// TIA Portal V18 export
FUNCTION_BLOCK "axis_FBD"   // FB53, FBD
{ S7_Optimized_Access := 'TRUE' }
VERSION : 0.1
// stored: AutoNumber true, IsIECCheckEnabled false, IsRetainMemResEnabled false, MemoryReserve 100, SetENOAutomatically false, UDAEnableTagReadback false
   VAR_INPUT
      "mm_per_ reductur outputshaft_rev (AskURmechEngineer)" : Real := 10.0;
      "reduction_ rotation (AskURmechEngineer)" : Real := 1.0;
      "ABincrements_per_ encoder_rev (CheckEnc Label and HSC hardware settings dont forget input filtration)" : Real := 4096.0;
      "max_revs_ at_10V (CheckMotorLabel)" : Real := 1360.0;
      "enc_placed_ on_motor not reductor output shaft(visually inspect)" : Bool;
      "isMultiturn (visually inspect)" : Bool;
      MultiTurnGoesFwdOnly : Bool;
      soft_speed_change_req : Bool;
      ENC_REVERSED_DIR : Bool;
      ENCODER_DINT : DInt;
      TargetUnison : Real;
      TargetHome : Real;
      Desk_bHome : Bool;
      Desk_bFwd : Bool;
      Desk_bRev : Bool;
      s_fwd_mechOK : Bool;
      s_rev_mecOK : Bool;
      s_fwd_ind : Bool;
      s_rev_ind : Bool;
      xPredifCal : Bool;
      ALIEN_MODE_EN : Bool;
      ALIEN_FWD : Bool;
      ALIEN_REV : Bool;
      ALIEN_SPDABS : Real;
      ExecUni : Bool;
      TheseAreDoors : Bool;
      xOverrideLocal : Bool;
      hbStepPlus : Bool;
      hbStepMinus : Bool;
      TargetStep : Real;
      динамические_границы_используются : Bool;
      динамическая_граница_fwd : Real;
      динамическая_граница_rev : Real;
   END_VAR
   VAR_OUTPUT
      max_speed_10V_p_mm : Real;
      speed_V : Real;
      speed : Real;
      yaINTSPEED : Int;
      yFWD : Bool;
      yREV : Bool;
      yFwd_STOP : Bool;
      yRev_STOP : Bool;
      yIN_POS : Bool;
      ER : Bool;
      WN : Bool;
      ALLOWED : Bool;
      "dist_stop(check t_acc)" : Real;
      MovingHomeWhileFree : Bool;
      ERWSTRING : WString;
   END_VAR
   VAR_IN_OUT
      aut_target : Real;
      para : "typeMotPara";
      POS : Real;
      calibrated : Bool;
      ENC_RET : "typePOSMEMcalib";
   END_VAR
   VAR
      para_ArtLimits { ExternalAccessible := 'False'; ExternalVisible := 'False'; ExternalWritable := 'False'} : "typeMotPara";
      v_absMax : Real;
      au_execute : Bool;
      AMANGRDB { S7_SetPoint := 'True'} : "axis_manager";
      MOTDB { S7_SetPoint := 'True'} : "__mot_universal_";
      WNDB { S7_SetPoint := 'True'} : "ER_WORD";
      ERDB { S7_SetPoint := 'True'} : "ER_WORD";
      erw_calcspd : WString;
      hmiResetCalib : Bool;
      IEC_Timer_0_Instance { S7_SetPoint := 'True'} : TON_TIME;
      artLimiter_Instance { S7_SetPoint := 'True'} : "artLimiter";
   END_VAR
   VAR_TEMP
      counts_per_mm : Real;
      er_params_mech : Bool;
      ENC : DInt;
      selected_man_speed : Real;
      AUTO : Bool;
      MAN : Bool;
      OVERRIDE : Bool;
      counts_real : Real;
      Enc_real_mm : Real;
      er_follow : Bool;
      er_set : Bool;
      er_fwd : Bool;
      er_rev : Bool;
      partners_calibrated : Bool;
      Selected_speed_auto : Real;
      ошибка_динамических_границ : Bool;
   END_VAR
BEGIN

REGION Network 1
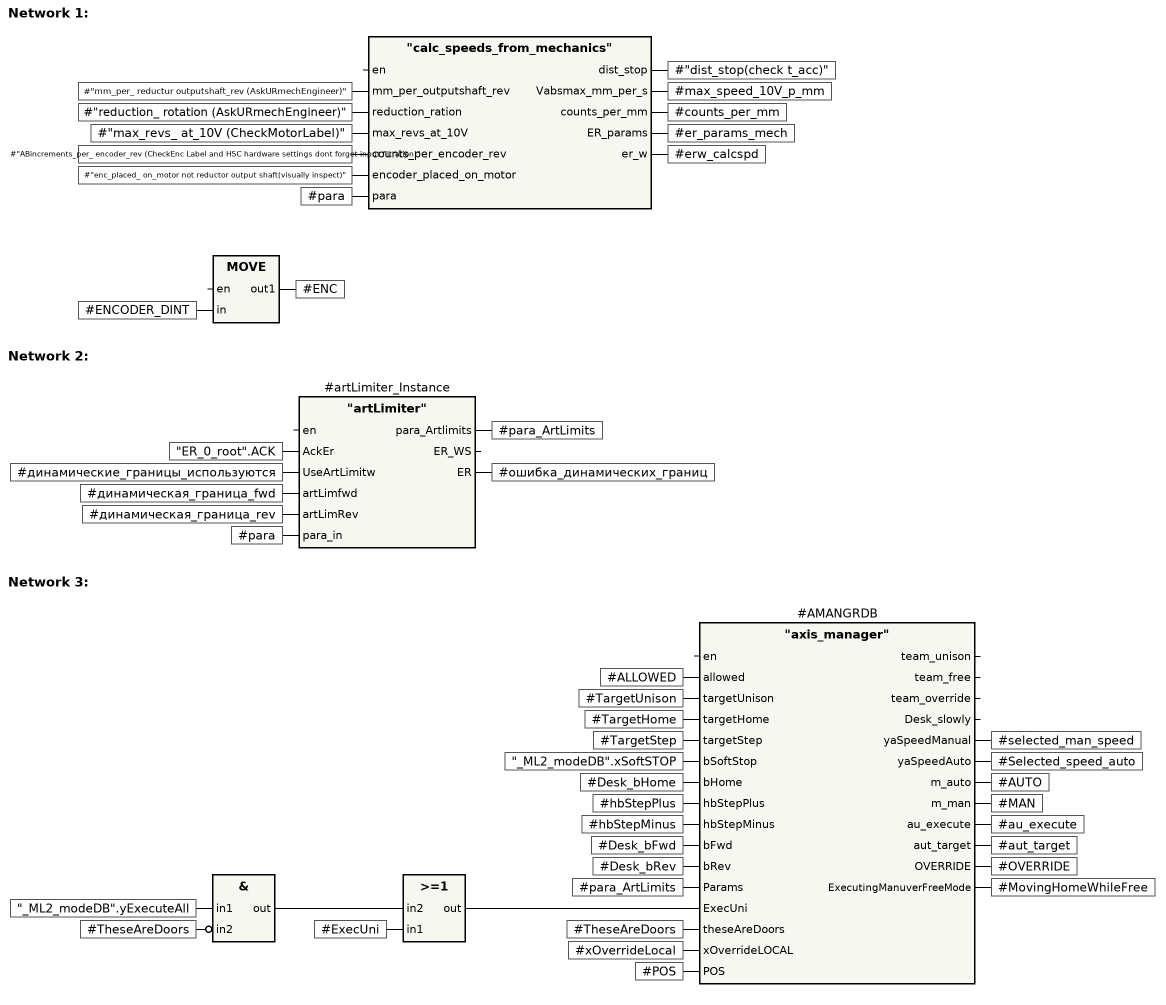
   "calc_speeds_from_mechanics"(mm_per_outputshaft_rev := #"mm_per_ reductur outputshaft_rev (AskURmechEngineer)",
                           reduction_ration := #"reduction_ rotation (AskURmechEngineer)",
                           max_revs_at_10V := #"max_revs_ at_10V (CheckMotorLabel)",
                           counts_per_encoder_rev := #"ABincrements_per_ encoder_rev (CheckEnc Label and HSC hardware settings dont forget input filtration)",
                           encoder_placed_on_motor := #"enc_placed_ on_motor not reductor output shaft(visually inspect)",
                           para := #para,
                           dist_stop => #"dist_stop(check t_acc)",
                           Vabsmax_mm_per_s => #max_speed_10V_p_mm,
                           counts_per_mm => #counts_per_mm,
                           ER_params => #er_params_mech,
                           er_w => #erw_calcspd);
   #ENC := #ENCODER_DINT;
END_REGION

REGION Network 2
   #artLimiter_Instance(AckEr := "ER_0_root".ACK,   // "artLimiter"
                        UseArtLimitw := #динамические_границы_используются,
                        artLimfwd := #динамическая_граница_fwd,
                        artLimRev := #динамическая_граница_rev,
                        para_in := #para,
                        para_Artlimits => #para_ArtLimits,
                        ER => #ошибка_динамических_границ);
END_REGION

REGION Network 3
   #AMANGRDB(allowed := #ALLOWED,   // "axis_manager"
             targetUnison := #TargetUnison,
             targetHome := #TargetHome,
             targetStep := #TargetStep,
             bSoftStop := "_ML2_modeDB".xSoftSTOP,
             bHome := #Desk_bHome,
             hbStepPlus := #hbStepPlus,
             hbStepMinus := #hbStepMinus,
             bFwd := #Desk_bFwd,
             bRev := #Desk_bRev,
             Params := #para_ArtLimits,
             ExecUni := ("_ML2_modeDB".yExecuteAll AND NOT #TheseAreDoors) OR #ExecUni,
             theseAreDoors := #TheseAreDoors,
             xOverrideLOCAL := #xOverrideLocal,
             POS := #POS,
             yaSpeedManual => #selected_man_speed,
             yaSpeedAuto => #Selected_speed_auto,
             m_auto => #AUTO,
             m_man => #MAN,
             au_execute => #au_execute,
             aut_target => #aut_target,
             OVERRIDE => #OVERRIDE,
             ExecutingManuverFreeMode => #MovingHomeWhileFree);
END_REGION

REGION Network 4 (SCL)

   ///1024 ppr, *4* mm per rev /10 reduction = mm
   //
   IF #ENC_REVERSED_DIR THEN
       #counts_real := - DINT_TO_REAL(#ENC);
   ELSE
       #counts_real := + DINT_TO_REAL(#ENC);
   END_IF;


   #Enc_real_mm :=  #counts_real / #counts_per_mm;
END_REGION

REGION Network 5
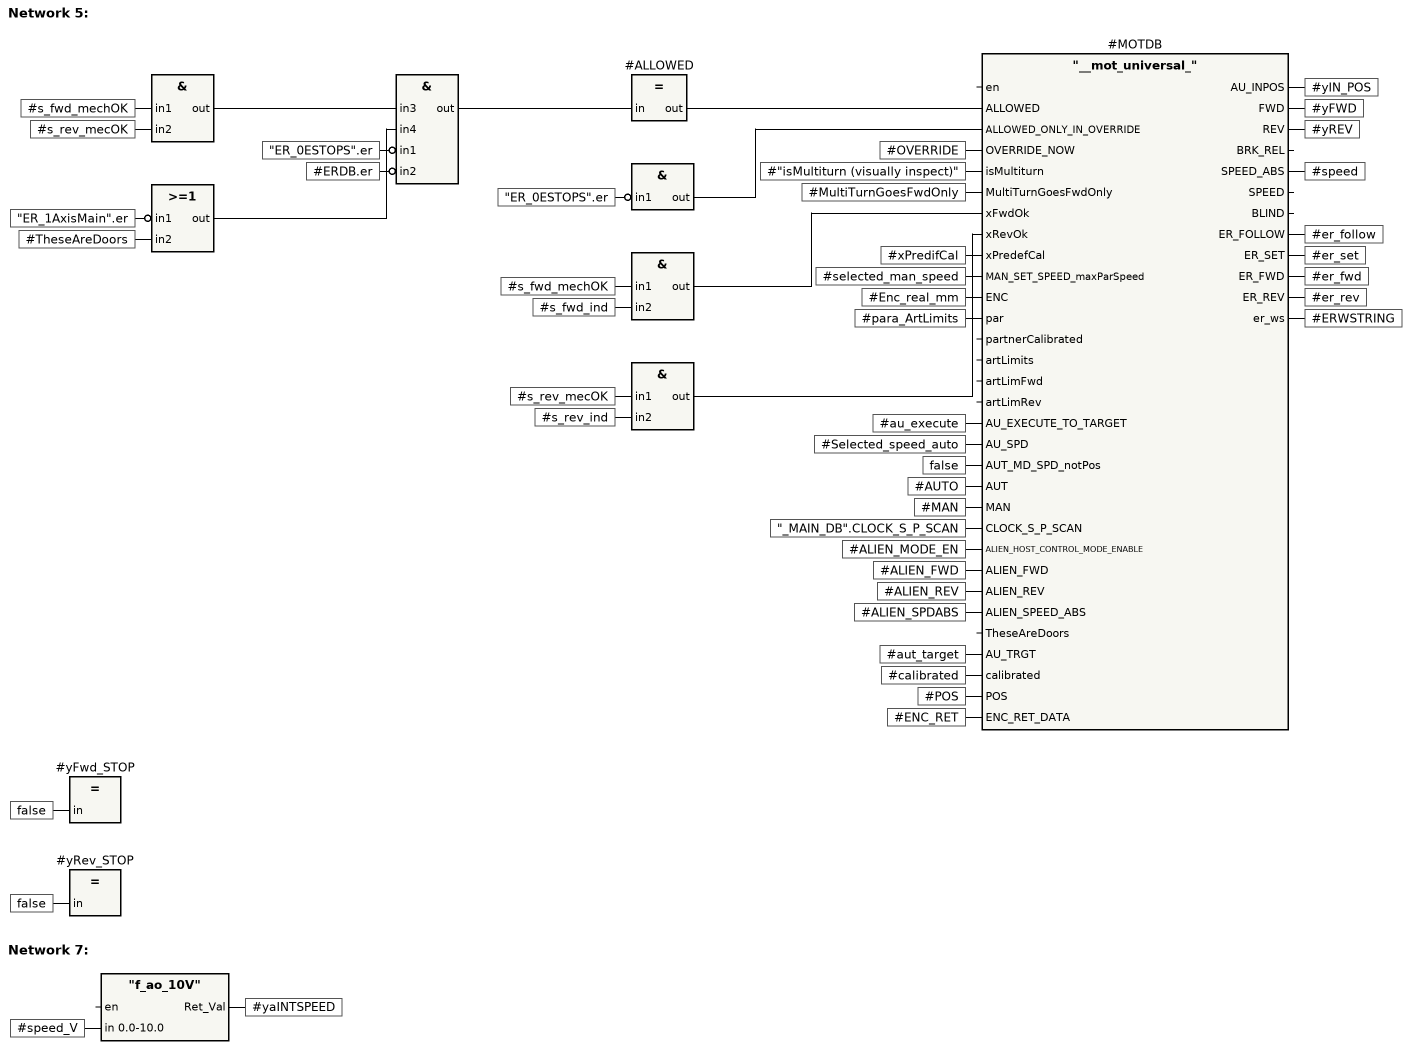
   #ALLOWED := #s_fwd_mechOK AND #s_rev_mecOK AND (NOT "ER_1AxisMain".er OR #TheseAreDoors) AND NOT "ER_0ESTOPS".er AND NOT #ERDB.er;
   #MOTDB(ALLOWED := #ALLOWED,   // "__mot_universal_"
          ALLOWED_ONLY_IN_OVERRIDE := NOT "ER_0ESTOPS".er,
          OVERRIDE_NOW := #OVERRIDE,
          isMultiturn := #"isMultiturn (visually inspect)",
          MultiTurnGoesFwdOnly := #MultiTurnGoesFwdOnly,
          xFwdOk := #s_fwd_mechOK AND #s_fwd_ind,
          xRevOk := #s_rev_mecOK AND #s_rev_ind,
          xPredefCal := #xPredifCal,
          MAN_SET_SPEED_maxParSpeed := #selected_man_speed,
          ENC := #Enc_real_mm,
          par := #para_ArtLimits,
          AU_EXECUTE_TO_TARGET := #au_execute,
          AU_SPD := #Selected_speed_auto,
          AUT_MD_SPD_notPos := false,
          AUT := #AUTO,
          MAN := #MAN,
          CLOCK_S_P_SCAN := "_MAIN_DB".CLOCK_S_P_SCAN,
          ALIEN_HOST_CONTROL_MODE_ENABLE := #ALIEN_MODE_EN,
          ALIEN_FWD := #ALIEN_FWD,
          ALIEN_REV := #ALIEN_REV,
          ALIEN_SPEED_ABS := #ALIEN_SPDABS,
          AU_TRGT := #aut_target,
          calibrated := #calibrated,
          POS := #POS,
          ENC_RET_DATA := #ENC_RET,
          AU_INPOS => #yIN_POS,
          FWD => #yFWD,
          REV => #yREV,
          SPEED_ABS => #speed,
          ER_FOLLOW => #er_follow,
          ER_SET => #er_set,
          ER_FWD => #er_fwd,
          ER_REV => #er_rev,
          er_ws => #ERWSTRING);
   #yFwd_STOP := false;
   #yRev_STOP := false;
END_REGION

REGION Network 6 (SCL)
   #speed_V := #speed / #max_speed_10V_p_mm * 10.0;
END_REGION

REGION Network 7
   #yaINTSPEED := "f_ao_10V"("in 0.0-10.0" := #speed_V);
END_REGION

REGION Network 8
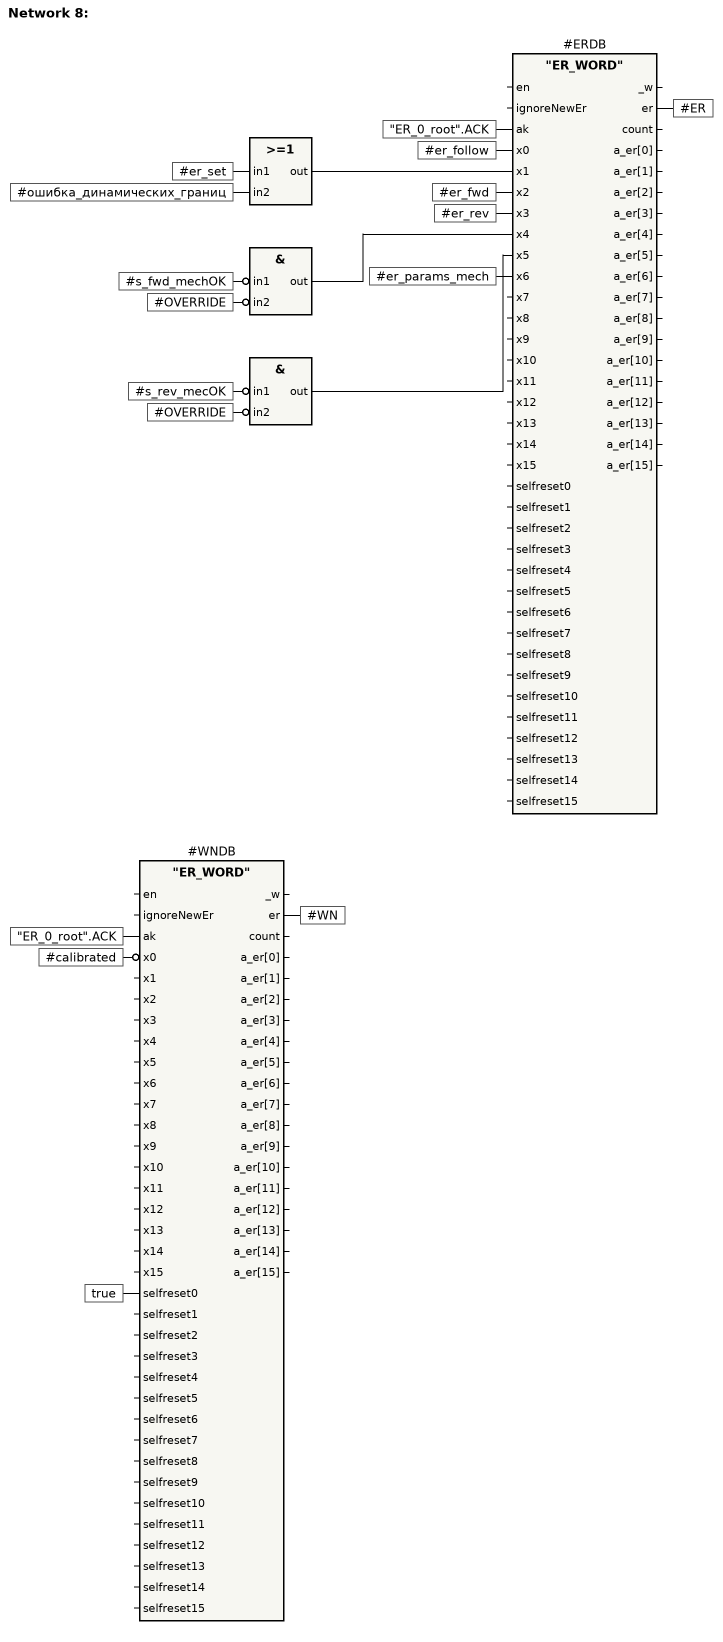
   #ERDB(ak := "ER_0_root".ACK,   // "ER_WORD"
         x0 := #er_follow,
         x1 := #er_set OR #ошибка_динамических_границ,
         x2 := #er_fwd,
         x3 := #er_rev,
         x4 := NOT #s_fwd_mechOK AND NOT #OVERRIDE,
         x5 := NOT #s_rev_mecOK AND NOT #OVERRIDE,
         x6 := #er_params_mech,
         er => #ER);
   #WNDB(ak := "ER_0_root".ACK, x0 := NOT #calibrated, selfreset0 := true, er => #WN);   // "ER_WORD"
END_REGION

REGION Network 9
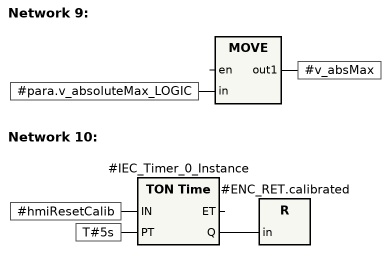
   #v_absMax := #para.v_absoluteMax_LOGIC;
END_REGION

REGION Network 10
   #IEC_Timer_0_Instance(IN := #hmiResetCalib, PT := T#5s);   // TON
   IF #IEC_Timer_0_Instance.Q THEN #ENC_RET.calibrated := FALSE; END_IF;
END_REGION
END_FUNCTION_BLOCK
